{attribute addProperty BoxType "EPP3744-0041-0016"}
{attribute addProperty Id "StatusAT %I*Status_F0C7FE3C1621ValueAT %I*DINT32417"}
{attribute addProperty CRC "1552041520"}
{attribute addProperty SizeInBites "48"}
{attribute addProperty SizeInBytes "6"}
TYPE AI_Inputs_Channel_5C824630 :
STRUCT
	{attribute addProperty Name "Status"}
	Status AT %I* : Status_F0C7FE3C;
	{attribute addProperty Name "Value"}
	Value AT %I* : DINT;
END_STRUCT
END_TYPE

(* stored: Version 1.2.0.0, ProductVersion 3.1.4024.9
   DUT AI_Inputs_Channel_5C824630: Id {6a083fba-1d86-40cd-ab34-6cd02e667827} *)
